(* IEC 61131-3 sources: teller/JD_Teller_LC2_V11/Class/Hub_Base, 1 file *)

(* ---- Hub_Base.st ---- *)
(*!
<Class
	Name               = "Hub_Base"
	Revision           = "1.20"
	RealtimeTask       = "false"
	CyclicTask         = "false"
	BackgroundTask     = "false"
	Sigmatek           = "true"
	OSInterface        = "false"
	HighPriority       = "false"
	Automatic          = "false"
	UpdateMode         = "Prescan"
	IconPath           = ".\Class\Tool.ico"
	SharedCommandTable = "true"
	Objectsize         = "(410,120)">
	<Channels>
		<Server Name="Control">
		</Server>
		<Client Name="Splitter_Place" Required="true" Internal="false" Comment="splitter place"/>
		<Client Name="VaranIn" Required="false" Internal="false"/>
	</Channels>
	<RevDoku>
		<Owner Company="Sigmatek" Author="renste"/>
		<Dokumentation Revision="1.20" Date="18.07.2013" Author="RamAnd" Company="Sigmatek" Description="Added NewInst forwarding"/>
		<Dokumentation Revision="1.15" Date="27.06.2011" Author="RamAnd" Company="Sigmatek" Description="Support of sorting VARAN commands by priority added (needed for communication between safety-modules)."/>
		<Dokumentation Revision="1.14" Date="04.01.2011" Author="BleErn" Company="Sigmatek" Description="Added Client Transparent that allows to disable a VARAN-HW-Class"/>
		<Dokumentation Revision="1.13" Date="14.10.2010" Author="RamAnd" Company="Sigmatek" Description="Added method AddMovDO for the move command in the VM."/>
		<Dokumentation Revision="1.12" Date="19.07.2010" Author="RamAnd" Company="Sigmatek" Description="Added new method GetNsTimeBPLLTicks for easier internal time measurements"/>
		<Dokumentation Revision="1.11" Date="31.05.2010" Author="BleErn" Company="Sigmatek" Description="Added support for RtPostScan"/>
		<Dokumentation Revision="1.10" Date="02.09.2009" Author="RamAnd" Company="Sigmatek" Description="Added functions for safety and hardware tree"/>
		<Dokumentation Revision="1.9" Date="16.07.2009" Author="ObeChr" Company="Sigmatek" Description="Added method: UseVaranRtPostScan"/>
		<Dokumentation Revision="1.8" Date="16.04.2009" Author="RamAnd" Company="Sigmatek" Description="Added 2 new methods: GetDocumentation and GetSerialNo"/>
	</RevDoku>
	<Network Name="Hub_Base">
		<!-- List of Components in this network -->
		<Components>
			<Object
				Name       = "_base"
				Class      = "VaranManager_Base"
				Position   = "(240,150)"
				Visualized = "true">
				<Channels>
					<Server Name="Control"/>
					<Client Name="To_FileSys"/>
					<Client Name="To_OSKernel"/>
					<Client Name="To_StdLib"/>
				</Channels>
			</Object>
		</Components>
		<Comments>
		</Comments>
		<!-- List of Connections in this network -->
		<Connections>
			<Connection Source="this.Control" Destination="_base.Control" Vertices="(712,210),(540,240),"/>
		</Connections>
		<!-- Headerfiles -->
		<Options>
		</Options>
	</Network>
</Class>
*)
#pragma using VaranManager_Base

Hub_Base : CLASS
: VaranManager_Base
  //Servers:
  //Clients:
	VaranIn 	: CltChCmd_Varan_Base;
	Splitter_Place 	: CltCh_DINT;
  //Variables:
  //Functions:
				//! <Function Comment="[#ENGLISH]&#13;&#10;=================================================================================================&#13;&#10;Function to add a realtime or cyclic task to VaranMaster&#13;&#10;=================================================================================================&#13;&#10;" Name="AddVaranTask"/>
	FUNCTION VIRTUAL GLOBAL AddVaranTask
		VAR_INPUT
			ud_dol_type 	: UDINT;			//! <Variable Comment=" Type of DOL (see lsl_st_varan.h)" Name="AddVaranTask.ud_dol_type"/>
			p_this 	: ^void;			//! <Variable Comment=" Thispointer of connected varan class" Name="AddVaranTask.p_this"/>
			callOptions 	: USINT := CALL_OPTION_RT_PRESCAN;
		END_VAR;
				//! <Function Comment="[#ENGLISH]&#13;&#10;=================================================================================================&#13;&#10;Function to add a read data object to varan master and install a varan task&#13;&#10;=================================================================================================&#13;&#10;" Name="AddRdDO"/>
	FUNCTION VIRTUAL GLOBAL AddRdDO
		VAR_INPUT
			p_us_position_info 	: ^USINT;			//! <Variable Comment="path of varan" Name="AddRdDO.p_us_position_info"/>
			ud_dol_type 	: UDINT;
			p_ud_handle 	: ^UDINT;			//! <Variable Comment=" pointer to variable to set right handle" Name="AddRdDO.p_ud_handle"/>
			ud_address 	: UDINT;			//! <Variable Comment="address to write" Name="AddRdDO.ud_address"/>
			ud_length 	: UDINT;			//! <Variable Comment="length of data (max. 128Byte)" Name="AddRdDO.ud_length"/>
			p_ud_data 	: ^UDINT;			//! <Variable Comment="pointer to data should be written" Name="AddRdDO.p_ud_data"/>
			ud_type 	: UDINT;			//! <Variable Comment="0=control area, 1=memory area" Name="AddRdDO.ud_type"/>
		END_VAR
		VAR_OUTPUT
			sd_retval 	: DINT;			//! <Variable Comment=" 0=OK, negative=error (look lsl_st_varan.h)" Name="AddRdDO.sd_retval"/>
		END_VAR;
				//! <Function Comment="[#ENGLISH]&#13;&#10;=================================================================================================&#13;&#10;Function to add a write data object to varan master and install a varan task&#13;&#10;=================================================================================================&#13;&#10;" Name="AddWrDO"/>
	FUNCTION VIRTUAL GLOBAL AddWrDO
		VAR_INPUT
			p_us_position_info 	: ^USINT;
			ud_dol_type 	: UDINT;
			p_ud_handle 	: ^UDINT;
			ud_address 	: UDINT;
			ud_length 	: UDINT;
			p_ud_data 	: ^UDINT;
			ud_type 	: UDINT;
		END_VAR
		VAR_OUTPUT
			sd_retval 	: DINT;
		END_VAR;
				//! <Function Comment="[#ENGLISH]&#13;&#10;=================================================================================================&#13;&#10;Function to add a read/write data object to varan master and install a varan task&#13;&#10;=================================================================================================&#13;&#10;" Name="AddRdWrDO"/>
	FUNCTION VIRTUAL GLOBAL AddRdWrDO
		VAR_INPUT
			p_us_position_info 	: ^USINT;
			ud_dol_type 	: UDINT;
			p_ud_handle 	: ^UDINT;
			ud_address_read 	: UDINT;			//! <Variable Comment=" Address of read data object" Name="AddRdWrDO.ud_address_read"/>
			ud_length_read 	: UDINT;			//! <Variable Comment=" Length of read data object" Name="AddRdWrDO.ud_length_read"/>
			p_ud_data_read 	: ^UDINT;			//! <Variable Comment=" pointer to variable to get pointer to data" Name="AddRdWrDO.p_ud_data_read"/>
			ud_address_write 	: UDINT;			//! <Variable Comment=" Address of write data object" Name="AddRdWrDO.ud_address_write"/>
			ud_length_write 	: UDINT;			//! <Variable Comment=" Length of write data object" Name="AddRdWrDO.ud_length_write"/>
			p_ud_data_write 	: ^UDINT;			//! <Variable Comment=" pointer to variable to get pointer to data" Name="AddRdWrDO.p_ud_data_write"/>
			ud_type 	: UDINT;
		END_VAR
		VAR_OUTPUT
			sd_retval 	: DINT;
		END_VAR;

	FUNCTION AWL VIRTUAL GLOBAL AddMovDO
		VAR_INPUT
			ud_dol_type 	: UDINT;
			p_ud_handle 	: ^UDINT;
			p_ud_MovSettings 	: ^UDINT;
			ud_type 	: UDINT;			//! <Variable Comment="access type is always memory, but we may want to have some priority for this access" Name="AddMovDO.ud_type"/>
		END_VAR
		VAR_OUTPUT
			sd_retval 	: DINT;
		END_VAR;
				//! <Function Comment="[#ENGLISH]&#13;&#10;=================================================================================================&#13;&#10;Function executes a data object list of VaranManager&#13;&#10;=================================================================================================&#13;&#10;" Name="ExecuteDOL"/>
	FUNCTION VIRTUAL GLOBAL ExecuteDOL
		VAR_INPUT
			ud_dol_type 	: UDINT;
		END_VAR
		VAR_OUTPUT
			sd_retval 	: DINT;
		END_VAR;
				//! <Function Comment="[#ENGLISH]&#13;&#10;=================================================================================================&#13;&#10;Function clears a data object list of VaranManager&#13;&#10;=================================================================================================&#13;&#10;" Name="ClearDOL"/>
	FUNCTION VIRTUAL GLOBAL ClearDOL
		VAR_INPUT
			ud_dol_type 	: UDINT;
		END_VAR
		VAR_OUTPUT
			sd_retval 	: DINT;
		END_VAR;
				//! <Function Comment="[#ENGLISH]&#13;&#10;=================================================================================================&#13;&#10;Function to read a direct access data object&#13;&#10;=================================================================================================&#13;&#10;" Name="RdDO"/>
	FUNCTION VIRTUAL GLOBAL RdDO
		VAR_INPUT
			p_us_position_info 	: ^USINT;
			ud_address 	: UDINT;
			ud_length 	: UDINT;
			p_ud_data 	: ^UDINT;
			ud_type 	: UDINT;
		END_VAR
		VAR_OUTPUT
			sd_retval 	: DINT;
		END_VAR;
				//! <Function Comment="[#ENGLISH]&#13;&#10;=================================================================================================&#13;&#10;Function to write a direct access data object&#13;&#10;=================================================================================================&#13;&#10;" Name="WrDO"/>
	FUNCTION VIRTUAL GLOBAL WrDO
		VAR_INPUT
			p_us_position_info 	: ^USINT;
			ud_address 	: UDINT;
			ud_length 	: UDINT;
			p_ud_data 	: ^UDINT;
			ud_type 	: UDINT;
		END_VAR
		VAR_OUTPUT
			sd_retval 	: DINT;
		END_VAR;
				//! <Function Comment="[#ENGLISH]&#13;&#10;=================================================================================================&#13;&#10;Function to get Pll - Time of VaranMaster&#13;&#10;=================================================================================================&#13;&#10;" Name="GetVaranTime"/>
	FUNCTION VIRTUAL GLOBAL GetVaranTime
		VAR_INPUT
			p_ud_IsoStartPoint 	: ^UDINT := NIL;
		END_VAR
		VAR_OUTPUT
			ud_varan_time 	: UDINT;			//! <Variable Comment=" Varantime in ns" Name="GetVaranTime.ud_varan_time"/>
		END_VAR;
				//! <Function Comment="[#ENGLISH]&#13;&#10;=================================================================================================&#13;&#10;Function to get Varan class position in a string&#13;&#10;=================================================================================================&#13;&#10;[local] p_us_node :W/R :help pointer to copy string&#13;&#10;" Name="GetVaranPosition"/>
	FUNCTION VIRTUAL GLOBAL GetVaranPosition
		VAR_INPUT
			p_us_info 	: ^USINT;			//! <Variable Comment=" pointer to save position info (first byte is length)" Name="GetVaranPosition.p_us_info"/>
		END_VAR
		VAR_OUTPUT
			sd_retval 	: DINT;
		END_VAR;
				//! <Function Comment="[#ENGLISH]&#13;&#10;=================================================================================================&#13;&#10;Function to install callback function for hot plug and play&#13;&#10;=================================================================================================&#13;&#10;" Name="SetObjectCallback"/>
	FUNCTION VIRTUAL GLOBAL SetObjectCallback
		VAR_INPUT
			p_us_position_info 	: ^USINT;
			ud_action_ptr 	: UDINT;			//! <Variable Comment="pointer to function" Name="SetObjectCallback.ud_action_ptr"/>
			ud_thisp 	: UDINT;			//! <Variable Comment="thispointer" Name="SetObjectCallback.ud_thisp"/>
			sd_required 	: DINT;			//! <Variable Comment="is class required" Name="SetObjectCallback.sd_required"/>
		END_VAR
		VAR_OUTPUT
			sd_retval 	: DINT;
		END_VAR;
				//! <Function Comment="[#ENGLISH]&#13;&#10;=================================================================================================&#13;&#10;Function sets Master off&#13;&#10;=================================================================================================&#13;&#10;" Name="SetManagerOff"/>
	FUNCTION VIRTUAL GLOBAL SetManagerOff
		VAR_INPUT
			e_error 	: t_e_VaranErrors;			//! <Variable Comment="reason why varan master is set off" Name="SetManagerOff.e_error"/>
		END_VAR;
				//! <Function Comment="[#ENGLISH]&#13;&#10;" Name="SetVaranError"/>
	FUNCTION VIRTUAL GLOBAL SetVaranError
		VAR_INPUT
			p_Node 	: ^USINT;			//! <Variable Comment="pointer to Node string" Name="SetVaranError.p_Node"/>
		END_VAR;
				//! <Function Comment="[#ENGLISH]&#13;&#10;=================================================================================================&#13;&#10;Function give back a nono second counter value of VaranMaster&#13;&#10;=================================================================================================&#13;&#10;" Name="GetNsTime"/>
	FUNCTION VIRTUAL GLOBAL GetNsTime
		VAR_OUTPUT
			ud_ns_counter 	: UDINT;			//! <Variable Comment="nano second counter value" Name="GetNsTime.ud_ns_counter"/>
		END_VAR;

	FUNCTION VIRTUAL GLOBAL GetNsTimeBPLLTicks
		VAR_OUTPUT
			ud_ns_counter 	: UDINT;			//! <Variable Comment="time since last tick" Name="GetNsTimeBPLLTicks.ud_ns_counter"/>
		END_VAR;
				//! <Function Comment="[#ENGLISH]&#13;&#10;=================================================================================================&#13;&#10;Function to get pointer to node information&#13;&#10;=================================================================================================&#13;&#10;" Name="GetNodeInfo"/>
	FUNCTION VIRTUAL GLOBAL GetNodeInfo
		VAR_INPUT
			p_us_position_info 	: ^USINT;
			p_node_info 	: ^PLSL_VARANNODEINFO;			//! <Variable Comment="pointer to node info" Name="GetNodeInfo.p_node_info"/>
		END_VAR
		VAR_OUTPUT
			sd_retval 	: DINT;
		END_VAR;
				//! <Function Comment="[#ENGLISH]&#13;&#10;=================================================================================================&#13;&#10;Function to get Varan Master number&#13;&#10;=================================================================================================&#13;&#10;[&lt;sd_master_number]number of varan master&#13;&#10;" Name="GetManagerNumber"/>
	FUNCTION VIRTUAL GLOBAL GetManagerNumber
		VAR_INPUT
			p_varan 	: ^pVoid;			//! <Variable Comment="address of pointer to varan" Name="GetManagerNumber.p_varan"/>
		END_VAR
		VAR_OUTPUT
			ud_manager_number 	: UDINT;
		END_VAR;
				//! <Function Comment="[#ENGLISH]&#13;&#10;=================================================================================================&#13;&#10;Function returns state of Varan manger class&#13;&#10;=================================================================================================&#13;&#10;" Name="GetManagerState"/>
	FUNCTION VIRTUAL GLOBAL GetManagerState
		VAR_OUTPUT
			e_state 	: t_e_VaranErrors;			//! <Variable Comment="error of varan manager" Name="GetManagerState.e_state"/>
		END_VAR;
				//! <Function Comment="[#ENGLISH]&#13;&#10;=================================================================================================&#13;&#10;Function to read SPI data&#13;&#10;=================================================================================================&#13;&#10;" Name="ReadSPIData"/>
	FUNCTION VIRTUAL GLOBAL ReadSPIData
		VAR_INPUT
			p_us_position_info 	: ^USINT;			//! <Variable Comment="nodestring of varan client" Name="ReadSPIData.p_us_position_info"/>
			ud_offset 	: UDINT;			//! <Variable Comment="offset in SPI flash" Name="ReadSPIData.ud_offset"/>
			ud_length 	: UDINT;			//! <Variable Comment="length of data to read (if MSB is set, access is done on the last page in SPI)" Name="ReadSPIData.ud_length"/>
			p_data 	: ^USINT;			//! <Variable Comment="pointer to allocated memory for read data" Name="ReadSPIData.p_data"/>
		END_VAR
		VAR_OUTPUT
			sd_retval 	: DINT;			//! <Variable Comment="0...success&#13;&#10;or else negative errorcode is returned" Name="ReadSPIData.sd_retval"/>
		END_VAR;
				//! <Function Comment="[#ENGLISH]&#13;&#10;=================================================================================================&#13;&#10;Function to get sync frame counter&#13;&#10;=================================================================================================&#13;&#10;" Name="GetSyncFrameCounter"/>
	FUNCTION VIRTUAL GLOBAL GetSyncFrameCounter
		VAR_OUTPUT
			us_frame_counter 	: USINT;			//! <Variable Comment=" sync frame counter" Name="GetSyncFrameCounter.us_frame_counter"/>
		END_VAR;
				//! <Function Comment="[#ENGLISH]&#13;&#10;=================================================================================================&#13;&#10;Function to log message&#13;&#10;=================================================================================================&#13;&#10;" Name="LogMessage"/>
	FUNCTION VIRTUAL GLOBAL LogMessage
		VAR_INPUT
			p_message 	: ^CHAR;			//! <Variable Comment="pointer to char string" Name="LogMessage.p_message"/>
			us_nr 	: USINT;			//! <Variable Comment="number of log variables" Name="LogMessage.us_nr"/>
			sd_var1 	: DINT;
			sd_var2 	: DINT;
			sd_var3 	: DINT;
		END_VAR;
				//! <Function Comment="[#DEUTSCH]&#13;&#10;=================================================================================================&#13;&#10;Function to disable device in cyclic&#13;&#10;=================================================================================================&#13;&#10;" Name="SetDisableDevice"/>
	FUNCTION VIRTUAL GLOBAL SetDisableDevice
		VAR_INPUT
			p_us_position_info 	: ^USINT;
		END_VAR
		VAR_OUTPUT
			sd_retval 	: DINT;
		END_VAR;

	FUNCTION VIRTUAL GLOBAL GetDocumentation
		VAR_INPUT
			p_us_position_info 	: ^USINT;
			p_dpne 	: ^CHAR;
		END_VAR
		VAR_OUTPUT
			sd_retval 	: DINT;
		END_VAR;

	FUNCTION VIRTUAL GLOBAL GetSerialNo
		VAR_INPUT
			p_us_position_info 	: ^USINT;
			p_SerialNo 	: ^CHAR;
		END_VAR
		VAR_OUTPUT
			sd_retval 	: DINT;
		END_VAR;

	FUNCTION VIRTUAL GLOBAL AllowRequiredError
		VAR_OUTPUT
			sd_retval 	: DINT;
		END_VAR;

	FUNCTION AWL VIRTUAL GLOBAL SetObjectThisp
		VAR_INPUT
			p_us_ObjectPath 	: ^USINT;
			ud_thisp 	: UDINT;
		END_VAR
		VAR_OUTPUT
			sd_retval 	: DINT;
		END_VAR;

	FUNCTION AWL VIRTUAL GLOBAL GetObjectThisp
		VAR_INPUT
			p_us_ObjectPath 	: ^USINT;
		END_VAR
		VAR_OUTPUT
			ud_thisp 	: UDINT;
		END_VAR;
				//! <Function Comment="[#ENGLISH]&#13;&#10;=================================================================================================&#13;&#10;Function to look if class is disabled&#13;&#10;=================================================================================================&#13;&#10;" Name="IsDeviceDisabled"/>
	FUNCTION VIRTUAL GLOBAL IsDeviceDisabled
		VAR_OUTPUT
			b_disabled 	: BOOL;			//! <Variable Comment="TRUE -&lt; Device disabled" Name="IsDeviceDisabled.b_disabled"/>
		END_VAR;

	FUNCTION VIRTUAL GLOBAL IsTransparent
		VAR_OUTPUT
			isTransparent 	: BOOL;
		END_VAR;

	FUNCTION VIRTUAL GLOBAL Control::NewInst
		VAR_INPUT
			pPara 	: ^CmdStruct;
			pResult 	: ^results;
		END_VAR
		VAR_OUTPUT
			ret_code 	: iprStates;
		END_VAR;
  //Tables:
	FUNCTION @STD
		VAR_OUTPUT
			ret_code	: CONFSTATES;
		END_VAR;
	FUNCTION GLOBAL TAB @CT_;
END_CLASS;

#pragma usingLtd Varan_Base

(************************************************************************************
*
*	Base class for Hubs
*	Created : Sigmatek	/	SR	/	March-April 2006
*	Changes :
*
*
*     FOR NEWER CHANGES SEE REVISION DOCUMENTATION IN CLASS PROPERTIES
*
*
*   1.6 => 1.7	/	26.05.2008
*			- [DB 863]: - add function to disable device in cyclic
*   1.5 => 1.6  /  18.04.2008
*			- [DB 852]: extend method GetVaranTime to get the IsoStartPoint
*		1.4 => 1.5	/ 	17.12.2007
*			- [DB 713]:	add function to log messages and log device error
*		1.3 => 1.4	/ 	03.10.2007
*			- add function to get "SyncFrame Counter"
*		1.2 => 1.3	/ 	04.04.2007
*			- [DB 541]: insert function to read SPI data
*		1.1 => 1.2	/	03.01.2007
*			[DB 418]: insert functions to disable and enable port
*		1.0 => 1.1	/ 	28.11.2006
*			first library version
*		0.2 => 1.0	/	05.10.2006
*			initial version
*		0.1 => 0.2	/	13.06.2006
*			second testversion
*		0.0	=> 0.1	/	10.04.2006
*			first testversion for fair in Hannover
*
************************************************************************************)

//[#ENGLISH]
//=================================================================================================
//Function to add a realtime or cyclic task to VaranMaster
//=================================================================================================
//[>ud_dol_type] type of DOL list( Realtime = 3, cyclic = 4 )
//[>p_this] Thispointer of connected varan class
FUNCTION VIRTUAL GLOBAL Hub_Base::AddVaranTask
	VAR_INPUT
		ud_dol_type 	: UDINT;
		p_this 	: ^void;
		callOptions 	: USINT;
	END_VAR

	VaranIn.VaranIn.AddVaranTask( ud_dol_type	:= ud_dol_type
								, p_this		:= p_this
                , callOptions := callOptions
								);

END_FUNCTION //VIRTUAL GLOBAL Hub_Base::AddVaranTask
//[#ENGLISH]
//=================================================================================================
//Function to add a read data object to varan master and install a varan task
//=================================================================================================
//[>p_us_position_info]pointer to position info( first byte is length)
//[>ud_dol_type] type of DOL list( 1=direct access, 2=IRQ, 3=realtime, 4=cyclic )
//[>p_ud_handle]pointer to variable to set right handle
//[>ud_address] Address of data object
//[>ud_length] Length of data object
//[>p_ud_data] pointer to variable to get pointer to data
//[>ud_type]0=control area, 1=memory area
//[<sd_retval] 0=OK, negative=error (look lsl_st_varan.h)
FUNCTION VIRTUAL GLOBAL Hub_Base::AddRdDO
VAR_INPUT
	p_us_position_info	: ^USINT;
	ud_dol_type			: UDINT;
	p_ud_handle			: ^UDINT;
	ud_address			: UDINT;
	ud_length			: UDINT;
	p_ud_data			: ^UDINT;
	ud_type				: UDINT;
END_VAR
VAR_OUTPUT
	sd_retval		: DINT;
END_VAR

	sd_retval := VaranIn.VaranIn.AddRdDO( p_us_position_info:= p_us_position_info
										, ud_dol_type		:= ud_dol_type
										, p_ud_handle		:= p_ud_handle
										, ud_address		:= ud_address
										, ud_length			:= ud_length
										, p_ud_data			:= p_ud_data
										, ud_type			:= ud_type
										);

END_FUNCTION //VIRTUAL GLOBAL Hub_Base::AddRdDO
//[#ENGLISH]
//=================================================================================================
//Function to add a write data object to varan master and install a varan task
//=================================================================================================
//[>p_us_position_info]pointer to position info( first byte is length)
//[>ud_dol_type] type of DOL list( 1=direct access, 2=IRQ, 3=realtime, 4=cyclic )
//[>p_ud_handle]pointer to variable to set right handle
//[>ud_address] Address of data object
//[>ud_length] Length of data object
//[>p_ud_data] pointer to variable to get pointer to data
//[>ud_type]0=control area, 1=memory area
//[<sd_retval] 0=OK, negative=error (look lsl_st_varan.h)
FUNCTION VIRTUAL GLOBAL Hub_Base::AddWrDO
VAR_INPUT
	p_us_position_info	: ^USINT;
	ud_dol_type			: UDINT;
	p_ud_handle			: ^UDINT;
	ud_address			: UDINT;
	ud_length			: UDINT;
	p_ud_data			: ^UDINT;
	ud_type				: UDINT;
END_VAR
VAR_OUTPUT
	sd_retval		: DINT;
END_VAR

	sd_retval := VaranIn.VaranIn.AddWrDO( p_us_position_info:= p_us_position_info
										, ud_dol_type		:= ud_dol_type
										, p_ud_handle		:= p_ud_handle
										, ud_address		:= ud_address
										, ud_length			:= ud_length
										, p_ud_data			:= p_ud_data
										, ud_type			:= ud_type
										);

END_FUNCTION //VIRTUAL GLOBAL Hub_Base::AddWrDO
//[#ENGLISH]
//=================================================================================================
//Function to add a read/write data object to varan master and install a varan task
//=================================================================================================
//[>p_us_position_info]pointer to position info( first byte is length)
//[>ud_dol_type] type of DOL list( 1=direct access, 2=IRQ, 3=realtime, 4=cyclic )
//[>p_ud_handle] pointer to variable to set right handle
//[>ud_address_read] Address of read data object
//[>ud_length_read] Length of read data object
//[>p_ud_data_read] pointer to variable to get pointer to data
//[>ud_address_write] Address of write data object
//[>ud_length_write] Length of write data object
//[>p_ud_data_write] pointer to variable to get pointer to data
//[>ud_type]0=control area, 1=memory area
//[<sd_retval] 0=OK, negative=error (look lsl_st_varan.h)
FUNCTION VIRTUAL GLOBAL Hub_Base::AddRdWrDO
VAR_INPUT
	p_us_position_info	: ^USINT;
	ud_dol_type			: UDINT;
	p_ud_handle			: ^UDINT;
	ud_address_read		: UDINT;
	ud_length_read		: UDINT;
	p_ud_data_read		: ^UDINT;
	ud_address_write	: UDINT;
	ud_length_write		: UDINT;
	p_ud_data_write		: ^UDINT;
	ud_type				: UDINT;
END_VAR
VAR_OUTPUT
	sd_retval		: DINT;
END_VAR

	sd_retval := VaranIn.VaranIn.AddRdWrDO	( p_us_position_info:= p_us_position_info
											, ud_dol_type		:= ud_dol_type
											, p_ud_handle		:= p_ud_handle
											, ud_address_read	:= ud_address_read
											, ud_length_read	:= ud_length_read
											, p_ud_data_read	:= p_ud_data_read
											, ud_address_write	:= ud_address_write
											, ud_length_write	:= ud_length_write
											, p_ud_data_write	:= p_ud_data_write
											, ud_type			:= ud_type
											);

END_FUNCTION //VIRTUAL GLOBAL Hub_Base::AddRdWrDO
//[#ENGLISH]
//=================================================================================================
//Function executes a data object list of VaranManager
//=================================================================================================
//[>ud_dol_type] type of DOL list( 1=direct access, 2=IRQ, 3=realtime, 4=cyclic )
//[<sd_retval] 0=OK, negative=error (look lsl_st_varan.h)
FUNCTION VIRTUAL GLOBAL Hub_Base::ExecuteDOL
VAR_INPUT
	ud_dol_type		: UDINT;
END_VAR
VAR_OUTPUT
	sd_retval		: DINT;
END_VAR

	sd_retval := VaranIn.VaranIn.ExecuteDOL( ud_dol_type := ud_dol_type );

END_FUNCTION //VIRTUAL GLOBAL Hub_Base::ExecuteDOL
//[#ENGLISH]
//=================================================================================================
//Function clears a data object list of VaranManager
//=================================================================================================
//[>ud_dol_type] Type of DOL (see lsl_st_varan.h)
//[<sd_retval] 0=OK, negative=error (look lsl_st_varan.h)
FUNCTION VIRTUAL GLOBAL Hub_Base::ClearDOL
VAR_INPUT
	ud_dol_type		: UDINT;
END_VAR
VAR_OUTPUT
	sd_retval		: DINT;
END_VAR

	sd_retval := VaranIn.VaranIn.ClearDOL( ud_dol_type := ud_dol_type );

END_FUNCTION //VIRTUAL GLOBAL Hub_Base::ClearDOL
//[#ENGLISH]
//=================================================================================================
//Function to read a direct access data object
//=================================================================================================
//[>p_us_position_info]pointer to position info( first byte is length)
//[>ud_address]address to read
//[>ud_length]length of data should read
//[>p_ud_data]variable to get pointer to readed data
//[>ud_type] 0=control area, 1=memory area
//[<sd_retval] 0=OK, negative=error (look lsl_st_varan.h)
FUNCTION VIRTUAL GLOBAL Hub_Base::RdDO
VAR_INPUT
	p_us_position_info	: ^USINT;
	ud_address			: UDINT;
	ud_length			: UDINT;
	p_ud_data			: ^UDINT;
	ud_type				: UDINT;
END_VAR
VAR_OUTPUT
	sd_retval			: DINT;
END_VAR

	sd_retval := VaranIn.VaranIn.RdDO	( p_us_position_info:= p_us_position_info
										, ud_address		:= ud_address
										, ud_length			:= ud_length
										, p_ud_data			:= p_ud_data
										, ud_type			:= ud_type
										);

END_FUNCTION //VIRTUAL GLOBAL Hub_Base::RdDO
//[#ENGLISH]
//=================================================================================================
//Function to write a direct access data object
//=================================================================================================
//[>p_us_position_info]pointer to position info( first byte is length)
//[>ud_address]address to write
//[>ud_length]length of data should be written
//[>p_ud_data]pointer to data should be written
//[>ud_type]0=control area, 1=memory area
//[<sd_retval] 0=OK, negative=error (look lsl_st_varan.h)
FUNCTION VIRTUAL GLOBAL Hub_Base::WrDO
VAR_INPUT
	p_us_position_info	: ^USINT;
	ud_address			: UDINT;
	ud_length			: UDINT;
	p_ud_data			: ^UDINT;
	ud_type				: UDINT;
END_VAR
VAR_OUTPUT
	sd_retval			: DINT;
END_VAR

	sd_retval := VaranIn.VaranIn.WrDO	( p_us_position_info:= p_us_position_info
										, ud_address		:= ud_address
										, ud_length			:= ud_length
										, p_ud_data			:= p_ud_data
										, ud_type			:= ud_type
										);

END_FUNCTION //VIRTUAL GLOBAL Hub_Base::WrDO
//[#ENGLISH]
//=================================================================================================
//Function to get Pll - Time of VaranMaster
//=================================================================================================
//[<ud_varan_time] Varantime in ns
FUNCTION VIRTUAL GLOBAL Hub_Base::GetVaranTime
VAR_INPUT
	p_ud_IsoStartPoint	: ^UDINT;
END_VAR
VAR_OUTPUT
	ud_varan_time		: UDINT;
END_VAR

	ud_varan_time := VaranIn.VaranIn.GetVaranTime( p_ud_IsoStartPoint );

END_FUNCTION //VIRTUAL GLOBAL Hub_Base::GetPllTime
//[#ENGLISH]
//=================================================================================================
//Function to get Varan class position in a string
//=================================================================================================
//[local]	p_us_node	:W/R	:help pointer to copy string
//[>p_us_info] pointer to save position info (first byte is length)
//[<sd_retval]0=OK, -1=to many hubs
FUNCTION VIRTUAL GLOBAL Hub_Base::GetVaranPosition
VAR_INPUT
	p_us_info		: ^USINT;
END_VAR
VAR_OUTPUT
	sd_retval		: DINT;
END_VAR
VAR
	p_us_node		: ^USINT;
END_VAR

#ifdef IsTransparent_IS_AVAILABLE
  IF VaranIn.IsTransparent() THEN
    IF Splitter_Place = 0 THEN
      // We can only forward on splitter place 0 - all other places would confuse the system...
      sd_retval := VaranIn.VaranIn.GetVaranPosition( p_us_info );
    ELSE
      sd_retval := -3;
    END_IF;
  ELSE
#endif

    sd_retval := 0;

    //if pointer is NIL do nothing
    if ( p_us_info <> NIL ) then

      p_us_node := VaranIn.GetPointer2NodeString();
      To_StdLib.MemCpy( dest 		:= p_us_info
              , source	:= p_us_node
              , size		:= p_us_node^ + 1
              );

      //increase length
      p_us_info^ += 1;

      //if max length is reached
      if ( p_us_info^ <= VARAN_MAX_DEPTH - 1 ) then

        //enter place on right position
        ( p_us_info + p_us_info^ )^ := TO_USINT( Splitter_Place );

      else
        sd_retval := -1;
      end_if;

    else
      sd_retval := -2;
    end_if;
#ifdef IsTransparent_IS_AVAILABLE
  END_IF;
#endif

END_FUNCTION //VIRTUAL GLOBAL Hub_Base::GetVaranPosition
//[#ENGLISH]
//=================================================================================================
//Function to install callback function for hot plug and play
//=================================================================================================
//[>p_us_position_info]pointer to position info( first byte is length)
//[>ud_action_ptr]pointer to function
//[>ud_thisp]thispointer
//[>sd_required]is class required
FUNCTION VIRTUAL GLOBAL Hub_Base::SetObjectCallback
VAR_INPUT
	p_us_position_info	: ^USINT;
	ud_action_ptr		: UDINT;
	ud_thisp			: UDINT;
	sd_required			: DINT;
END_VAR
VAR_OUTPUT
	sd_retval		: DINT;
END_VAR

	sd_retval := VaranIn.VaranIn.SetObjectCallback	( p_us_position_info:= p_us_position_info
													, ud_action_ptr		:= ud_action_ptr
													, ud_thisp			:= ud_thisp
													, sd_required		:= sd_required
													);

END_FUNCTION //VIRTUAL GLOBAL Hub_Base::SetObjectCallback
//[#ENGLISH]
//=================================================================================================
//Function sets Master off
//=================================================================================================
//[>e_error]reason why varan master is set off
FUNCTION VIRTUAL GLOBAL Hub_Base::SetManagerOff
VAR_INPUT
	e_error	: t_e_VaranErrors;
END_VAR

	VaranIn.VaranIn.SetManagerOff( e_error := e_error );

END_FUNCTION //VIRTUAL GLOBAL Hub_Base::SetMasterOff
//[#ENGLISH]
//[>p_Node]pointer to Node string
FUNCTION VIRTUAL GLOBAL Hub_Base::SetVaranError
VAR_INPUT
	p_Node		: ^USINT;
END_VAR

	VaranIn.VaranIn.SetVaranError( p_Node := p_Node );

END_FUNCTION //VIRTUAL GLOBAL Hub_Base::SetVaranError
//[#ENGLISH]
//=================================================================================================
//Function give back a nono second counter value of VaranMaster
//=================================================================================================
//[<ud_ns_counter]nano second counter value
FUNCTION VIRTUAL GLOBAL Hub_Base::GetNsTime
VAR_OUTPUT
	ud_ns_counter		: UDINT;
END_VAR

	ud_ns_counter := VaranIn.VaranIn.GetNsTime();

END_FUNCTION //VIRTUAL GLOBAL Hub_Base::GetNsTime
//[#ENGLISH]
//=================================================================================================
//Function to get pointer to node information
//=================================================================================================
//[>p_us_position_info]pointer to position info( first byte is length)
//[>p_node_info]pointer to node info
FUNCTION VIRTUAL GLOBAL Hub_Base::GetNodeInfo
VAR_INPUT
	p_us_position_info		: ^USINT;
	p_node_info		: ^PLSL_VARANNODEINFO;
END_VAR
VAR_OUTPUT
	sd_retval		: DINT;
END_VAR

	sd_retval := VaranIn.VaranIn.GetNodeInfo( p_us_position_info	:= p_us_position_info
											, p_node_info			:= p_node_info
											);

END_FUNCTION //VIRTUAL GLOBAL Hub_Base::GetNodeInfo
//[#ENGLISH]
//=================================================================================================
//Function to get Varan Master number
//=================================================================================================
//[<sd_master_number]number of varan master
//[>p_varan]address of pointer to varan
FUNCTION VIRTUAL GLOBAL Hub_Base::GetManagerNumber
VAR_INPUT
	p_varan				: ^pVoid;
END_VAR
VAR_OUTPUT
	ud_manager_number	: UDINT;
END_VAR

	ud_manager_number := VaranIn.VaranIn.GetManagerNumber( p_varan := p_varan );

END_FUNCTION //VIRTUAL GLOBAL Hub_Base::GetMasterNumber
//[#ENGLISH]
//=================================================================================================
//Function returns state of Varan manger class
//=================================================================================================
//[<e_state]error of varan manager
FUNCTION VIRTUAL GLOBAL Hub_Base::GetManagerState
VAR_OUTPUT
	e_state		: t_e_VaranErrors;
END_VAR

	e_state := VaranIn.VaranIn.GetManagerState();

END_FUNCTION //VIRTUAL GLOBAL Hub_Base::GetManagerState
//[#ENGLISH]
//=================================================================================================
//Function to look if class is disabled
//=================================================================================================
//[<b_disabled]TRUE -< Device disabled
FUNCTION VIRTUAL GLOBAL Hub_Base::IsDeviceDisabled
VAR_OUTPUT
	b_disabled		: BOOL;
END_VAR

	b_disabled := VaranIn.IsDeviceDisabled();

END_FUNCTION //VIRTUAL GLOBAL Hub_Base::IsDeviceDisabled
//[#ENGLISH]
//=================================================================================================
//Function to read SPI data
//=================================================================================================
//[>p_us_position_info]pointer to position info( first byte is length)
//[>ud_offset]offset in SPI flash
//[>ud_length]length of data (max. 128Byte)
//[>p_data]pointer to allocated memory for read data
//[<sd_retval] 0=OK, negative=error (look lsl_st_varan.h)
FUNCTION VIRTUAL GLOBAL Hub_Base::ReadSPIData
VAR_INPUT
	p_us_position_info	: ^USINT;
	ud_offset			: UDINT;
	ud_length			: UDINT;
	p_data				: ^USINT;
END_VAR
VAR_OUTPUT
	sd_retval		: DINT;
END_VAR

	sd_retval := VaranIn.VaranIn.ReadSPIData( p_us_position_info	:= p_us_position_info
											, ud_offset				:= ud_offset
											, ud_length				:= ud_length
											, p_data 				:= p_data
											);

END_FUNCTION //VIRTUAL GLOBAL Hub_Base::ReadSPIData
//[#ENGLISH]
//=================================================================================================
//Function to get sync frame counter
//=================================================================================================
//[<us_frame_counter] sync frame counter
FUNCTION VIRTUAL GLOBAL Hub_Base::GetSyncFrameCounter
VAR_OUTPUT
	us_frame_counter		: USINT;
END_VAR

	us_frame_counter := VaranIn.VaranIn.GetSyncFrameCounter();

END_FUNCTION //VIRTUAL GLOBAL Hub_Base::GetSyncFramCounter
//[#ENGLISH]
//=================================================================================================
//Function to log message
//=================================================================================================
//[>p_message]pointer to char string
//[>us_nr]number of log variables
FUNCTION VIRTUAL GLOBAL Hub_Base::LogMessage
VAR_INPUT
	p_message	: ^CHAR;
	us_nr		: USINT;
	sd_var1		: DINT;
	sd_var2		: DINT;
	sd_var3		: DINT;
END_VAR

	VaranIn.VaranIn.LogMessage	( p_message	:= p_message
								, us_nr		:= us_nr
								, sd_var1	:= sd_var1
								, sd_var2	:= sd_var2
								, sd_var3	:= sd_var3
								);

END_FUNCTION //VIRTUAL GLOBAL Hub_Base::LogMessage
//[#DEUTSCH]
//=================================================================================================
//Function to disable device in cyclic
//=================================================================================================
//[>p_us_position_info]path of varan
FUNCTION VIRTUAL GLOBAL Hub_Base::SetDisableDevice
VAR_INPUT
	p_us_position_info		: ^USINT;
END_VAR
VAR_OUTPUT
	sd_retval		: DINT;
END_VAR

	sd_retval := VaranIn.VaranIn.SetDisableDevice( p_us_position_info := p_us_position_info );

END_FUNCTION //VIRTUAL GLOBAL Hub_Base::SetDisableDevice

FUNCTION VIRTUAL GLOBAL Hub_Base::GetDocumentation
	VAR_INPUT
		p_us_position_info 	: ^USINT;
		p_dpne 	: ^CHAR;
	END_VAR
	VAR_OUTPUT
		sd_retval 	: DINT;
	END_VAR

  sd_retval := VaranIn.VaranIn.GetDocumentation(p_us_position_info, p_dpne);

END_FUNCTION

FUNCTION VIRTUAL GLOBAL Hub_Base::GetSerialNo
	VAR_INPUT
		p_us_position_info 	: ^USINT;
		p_SerialNo 	: ^CHAR;
	END_VAR
	VAR_OUTPUT
		sd_retval 	: DINT;
	END_VAR

  sd_retval := VaranIn.VaranIn.GetSerialNo(p_us_position_info, p_SerialNo);

END_FUNCTION

FUNCTION VIRTUAL GLOBAL Hub_Base::AllowRequiredError
	VAR_OUTPUT
		sd_retval 	: DINT;
	END_VAR

  sd_retval := VaranIn.VaranIn.AllowRequiredError();

END_FUNCTION

FUNCTION VIRTUAL GLOBAL Hub_Base::SetObjectThisp
	VAR_INPUT
		p_us_ObjectPath 	: ^USINT;
		ud_thisp 	: UDINT;
	END_VAR
	VAR_OUTPUT
		sd_retval 	: DINT;
	END_VAR

  sd_retval := VaranIn.VaranIn.SetObjectThisp(p_us_ObjectPath:=p_us_ObjectPath, ud_thisp:=ud_thisp);

END_FUNCTION

FUNCTION VIRTUAL GLOBAL Hub_Base::GetObjectThisp
	VAR_INPUT
		p_us_ObjectPath 	: ^USINT;
	END_VAR
	VAR_OUTPUT
		ud_thisp 	: UDINT;
	END_VAR

  ud_thisp := VaranIn.VaranIn.GetObjectThisp(p_us_ObjectPath:=p_us_ObjectPath);

END_FUNCTION

FUNCTION VIRTUAL GLOBAL Hub_Base::GetNsTimeBPLLTicks
	VAR_OUTPUT
		ud_ns_counter 	: UDINT;
	END_VAR

  ud_ns_counter := VaranIn.VaranIn.GetNsTimeBPLLTicks();

END_FUNCTION

FUNCTION VIRTUAL GLOBAL Hub_Base::AddMovDO
	VAR_INPUT
		ud_dol_type 	: UDINT;
		p_ud_handle 	: ^UDINT;
		p_ud_MovSettings 	: ^UDINT;
		ud_type 	: UDINT;
	END_VAR
	VAR_OUTPUT
		sd_retval 	: DINT;
	END_VAR

  sd_retval := VaranIn.VaranIn.AddMovDO(ud_dol_type:=ud_dol_type
                                      , p_ud_handle:=p_ud_handle
                                      , p_ud_MovSettings:=p_ud_MovSettings
                                      , ud_type:=ud_type);

END_FUNCTION

FUNCTION VIRTUAL GLOBAL Hub_Base::IsTransparent
	VAR_OUTPUT
		isTransparent 	: BOOL;
	END_VAR

#ifdef IsTransparent_IS_AVAILABLE
  IF VaranIn.IsTransparent() & Splitter_Place = 0 THEN
    isTransparent := VaranIn.VaranIn.IsTransparent();
  ELSE
    isTransparent := VaranIn.IsTransparent();
  END_IF;
#else
  isTransparent := FALSE;
#endif

END_FUNCTION

FUNCTION VIRTUAL GLOBAL Hub_Base::Control::NewInst
	VAR_INPUT
		pPara 	: ^CmdStruct;
		pResult 	: ^Results;
	END_VAR
	VAR_OUTPUT
		ret_code 	: IprStates;
	END_VAR

	ret_code := VaranIn.VaranIn.NewInst(pPara, pResult);

END_FUNCTION
